// TwinCAT 3 PLC project FMFiles
// Title: FM Files
// Company: FrameworkMonorepo
// ProjectVersion: 0.0.1
// ProgramVersion: 3.1.4024.0
// libraries:
//   FM Common Interfaces, * (FrameworkMonorepo)
//   FM Events, * (FrameworkMonorepo)
//   FM Strings, * (FrameworkMonorepo)
//   Tc2_Standard, * (Beckhoff Automation GmbH)
//   Tc2_System, * (Beckhoff Automation GmbH)
//   Tc2_Utilities, * (Beckhoff Automation GmbH)
// project tree:
//   File/ Directory.TcPOU, File.TcPOU, FileRemover.TcPOU
//   Version/ Global_Version.TcGVL
// (motion and I/O tree: see PLC project fmtypes)
// real-time tasks:
//   TASK BindingTestTask: cycle T#1ms, priority 20, ADS port 350
//   TASK PlcTask: cycle T#1ms, priority 21, ADS port 351
//   TASK PlcTask1: cycle T#1ms, priority 22, ADS port 352
//   TASK PlcTask2: cycle T#1ms, priority 23, ADS port 353
//   TASK MathTestTask: cycle T#1ms, priority 24, ADS port 354
//   TASK TimesTestsTask: cycle T#1ms, priority 25, ADS port 355

// ---- Version/Global_Version.TcGVL
{attribute 'TcGenerated'}
{attribute 'no-analysis'}
{attribute 'linkalways'}
// This function has been automatically generated from the project information.
VAR_GLOBAL CONSTANT
	{attribute 'const_non_replaced'}
	stLibVersion_FM_Files : ST_LibVersion := (iMajor := 0, iMinor := 0, iBuild := 1, iRevision := 0, nFlags := 0, sVersion := '0.0.1');
END_VAR

// ---- File/Directory.TcPOU
FUNCTION_BLOCK Directory
VAR
	creator : FB_CreateDir; // can only create on level of folder
	remover : FB_RemoveDir; // can only remove topmost folder. Not folder with folders.

	listDir : FB_EnumFindFileList;	
	listing : BOOL;
	_ListDone : BOOL;
	checkingFolder : BOOL;
	checkingFileExistence : BOOL;

	page : ARRAY[0..50 - 1] OF ST_FindFileEntry;
	_FileNameList : ARRAY[0..50 - 1] OF T_MaxString;
	_FileExists : BOOL;
	
	filenameForAlarm : T_MaxString;
	createDirectoryErrorTrig : R_TRIG;
	removeDirectoryErrorTrig : R_TRIG;
	listingDirectoryErrorTrig : R_TRIG;
	createDirectoryError : MessageEventLogger(TC_EVENTS.DirectoryEventClass.CreateDirectoryError);
	removeDirectoryError : MessageEventLogger(TC_EVENTS.DirectoryEventClass.RemoveDirectoryError);
	listingDirectoryError : MessageEventLogger(TC_EVENTS.DirectoryEventClass.ListDirectoryError);
END_VAR
VAR CONSTANT
	EntriesPerPage : INT := 50;
END_VAR

METHOD PRIVATE Abort
VAR_INPUT
END_VAR
listDir(
	bExecute := TRUE,
	eCmd := E_EnumCmdType.eEnumCmd_Abort
);
listDir(bExecute := FALSE);
END_METHOD

{attribute 'TcRpcEnable':='1'}
METHOD Create
VAR_INPUT
	path : T_MaxString;
END_VAR
creator(
	sPathName := path,
	bExecute := TRUE,
);
END_METHOD

METHOD Cyclic
VAR
	i : INT;
END_VAR
creator(bExecute := FALSE);
remover(bExecute := FALSE);

listDir(
	pFindList := ADR(page),
	cbFindList := SIZEOF(page)
);

IF (NOT listDir.bBusy AND listing AND NOT _ListDone AND listDir.eCmd <> E_EnumCmdType.eEnumCmd_Abort) THEN

	listDir(bExecute := FALSE);
	listing := FALSE;
	_ListDone := TRUE;
	
	FOR i := 0 TO EntriesPerPage - 1 DO
		_FileNameList[i] := page[i].sFileName;
		
		IF (checkingFileExistence) THEN
			IF (page[i].fileAttributes.bDirectory = checkingFolder
				AND page[i].sFileName <> '') THEN
				_FileExists := TRUE;
			END_IF
		END_IF
	END_FOR
	
	IF (NOT listDir.bEOE) THEN
		Abort();
	END_IF
END_IF

createDirectoryErrorTrig(CLK := creator.bError);
removeDirectoryErrorTrig(CLK := remover.bError);
listingDirectoryErrorTrig(CLK := listDir.bError);

IF (createDirectoryErrorTrig.Q) THEN
	filenameForAlarm := creator.sPathName;
	IF (EventParameters.EscapeBackslash) THEN
		filenameForAlarm := ReplaceAll(filenameForAlarm, '\', '\\'); // Escape backslash to use with web-based HMIs
	END_IF
	createDirectoryError.Arguments.Clear().AddStringByValue(filenameForAlarm);
	createDirectoryError.Send();
END_IF
IF (removeDirectoryErrorTrig.Q) THEN
	filenameForAlarm := remover.sPathName;
	IF (EventParameters.EscapeBackslash) THEN
		filenameForAlarm := ReplaceAll(filenameForAlarm, '\', '\\'); // Escape backslash to use with web-based HMIs
	END_IF
	removeDirectoryError.Arguments.Clear().AddStringByValue(filenameForAlarm);
	removeDirectoryError.Send();
END_IF
IF (listingDirectoryErrorTrig.Q) THEN
	filenameForAlarm := listDir.sPathName;
	IF (EventParameters.EscapeBackslash) THEN
		filenameForAlarm := ReplaceAll(filenameForAlarm, '\', '\\'); // Escape backslash to use with web-based HMIs
	END_IF
	listingDirectoryError.Arguments.Clear().AddStringByValue(filenameForAlarm);
	listingDirectoryError.Send();
END_IF
END_METHOD

{attribute 'monitoring' := 'call'}
PROPERTY FileExists : BOOL
GET
FileExists := _FileExists;
END_GET
END_PROPERTY

{attribute 'monitoring' := 'call'}
PROPERTY FileNameList : REFERENCE TO ARRAY[0..49] OF T_MaxString
GET
FileNameList REF= _FileNameList;
END_GET
END_PROPERTY

METHOD CheckFileExists
VAR_INPUT
	path : T_MaxString;
	folder : BOOL; // FALSE = File, TRUE = Folder
END_VAR
IF (NOT listDir.bBusy) THEN
	
	List(path);
	
	_FileExists := FALSE;
	checkingFileExistence := TRUE;
	checkingFolder := folder;
END_IF
END_METHOD

 // Usage of * wildcard recommended
 // Add * to the end of path to list all files
METHOD List
VAR_INPUT
	path : T_MaxString;
END_VAR
IF (NOT listDir.bBusy) THEN
	
	checkingFileExistence := FALSE;
	listing := TRUE;
	_ListDone := FALSE;
	
	listDir(bExecute := FALSE);
	listDir(
		sPathName := path,
		eCmd := E_EnumCmdType.eEnumCmd_First,
		bExecute := TRUE
	);
END_IF
END_METHOD

PROPERTY ListDone : BOOL
GET
ListDone := _ListDone;
END_GET
END_PROPERTY

METHOD Remove
VAR_INPUT
	path : T_MaxString;
END_VAR
remover(
	sPathName := path,
	bExecute := TRUE,
);
END_METHOD

END_FUNCTION_BLOCK

// ---- File/File.TcPOU
FUNCTION_BLOCK File IMPLEMENTS Cyclic
VAR
	_Busy : BOOL;
	_Done : BOOL;
	_Error : BOOL;
	
	openRequest : BOOL;
	readRequest : BOOL;
	writeRequest : BOOL;
	appendMode : BOOL;
	filePath : T_MaxString;
	
	buffer : POINTER TO BYTE;
	bufferLength : UDINT;

	handle : UINT;
	opener : FB_FileOpen;
	closer : FB_FileClose;
	reader : FB_FileRead;
	writer : FB_FileWrite;
	
	fileState : (Waiting, OpenMode, Opening, Reading, Writing, Closing);
	
	filenameForAlarm : T_MaxString;
	openErrorTrigger : R_TRIG;
	readErrorTrigger : R_TRIG;
	writeErrorTrigger : R_TRIG;
	closeErrorTrigger : R_TRIG;
	notFoundError : MessageEventLogger(TC_EVENTS.FileEventClass.InvalidPath);
	fileOpenError : MessageEventLogger(TC_EVENTS.FileEventClass.OpenFileError);
	fileReadError : MessageEventLogger(TC_EVENTS.FileEventClass.ReadFileError);
	fileWriteError : MessageEventLogger(TC_EVENTS.FileEventClass.WriteFileError);
	fileCloseError : MessageEventLogger(TC_EVENTS.FileEventClass.CloseFileError);
END_VAR
VAR CONSTANT
	NotFoundErrorNumber : UDINT := 16#70C;
END_VAR

{attribute 'monitoring' := 'call'}
PROPERTY Busy : BOOL
GET
Busy := _Busy;
END_GET
END_PROPERTY

METHOD Cyclic
CASE fileState OF
	
	Waiting:
	
		IF (openRequest) THEN
			openRequest := FALSE;
			_Done := FALSE;
			
			fileState := OpenMode;
		END_IF
	
	OpenMode:
	
		IF (readRequest) THEN
			opener.nMode := FOPEN_MODEREAD;
		ELSIF (writeRequest) THEN
			IF (appendMode) THEN
				opener.nMode := FOPEN_MODEAPPEND;
			ELSE
				opener.nMode := FOPEN_MODEWRITE;
			END_IF
		END_IF
		
		opener.nMode := opener.nMode OR FOPEN_MODETEXT;

		fileState := Opening;
	
	Opening:
	
		opener(
			bExecute := NOT opener.bBusy,
			sPathName := filePath,
			hFile => handle,
		);
		
		IF (NOT opener.bExecute AND NOT opener.bBusy AND handle <> 0) THEN
			opener();
			IF (readRequest) THEN
				fileState := Reading;
			ELSIF (writeRequest) THEN
				fileState := Writing;
			END_IF
		END_IF
	
	Reading:
	
		reader(
			bExecute := NOT reader.bBusy,
			hFile := handle,
			pReadBuff := buffer,
			cbReadLen := bufferLength,
		);
		
		IF (NOT reader.bExecute AND NOT reader.bBusy) THEN
			fileState := Closing;
		END_IF
	
	Writing:
	
		writer(
			bExecute := NOT writer.bBusy,
			hFile := handle,
			pWriteBuff := buffer,
			cbWriteLen := bufferLength,
		);
		
		IF (NOT writer.bExecute AND NOT writer.bBusy) THEN
			fileState := Closing;
		END_IF
	
	Closing:
	
		IF (handle = 0) THEN
			fileState := Waiting;
		ELSE
			closer(
				bExecute := NOT closer.bBusy,
				hFile := handle,
			);
			
			IF (NOT closer.bExecute AND NOT closer.bBusy) THEN
				closer();
				handle := 0;
				_Done := TRUE;
				
				fileState := Waiting;
			END_IF
		END_IF
	
END_CASE

_Busy := fileState <> Waiting;

openErrorTrigger(CLK := opener.bError);
readErrorTrigger(CLK := reader.bError);
writeErrorTrigger(CLK := writer.bError);
closeErrorTrigger(CLK := closer.bError);
_Error := 
	openErrorTrigger.Q
	OR readErrorTrigger.Q
	OR writeErrorTrigger.Q
	OR closeErrorTrigger.Q
	;
IF (_Error) THEN
	openRequest := FALSE;
	readRequest := FALSE;
	writeRequest := FALSE;
	
	filenameForAlarm := opener.sPathName;
	IF (EventParameters.EscapeBackslash) THEN
		filenameForAlarm := ReplaceAll(filenameForAlarm, '\', '\\'); // Escape backslash to use with web-based HMIs
	END_IF
	
	IF (openErrorTrigger.Q AND opener.nErrId = NotFoundErrorNumber) THEN
		notFoundError.Arguments.Clear().AddStringByValue(filenameForAlarm);
		notFoundError.Send();
	ELSIF (openErrorTrigger.Q) THEN
		fileOpenError.Arguments.Clear().AddStringByValue(filenameForAlarm);
		fileOpenError.Send();
	ELSIF (readErrorTrigger.Q) THEN
		fileReadError.Arguments.Clear().AddStringByValue(filenameForAlarm);
		fileReadError.Send();
	ELSIF (openErrorTrigger.Q) THEN
		fileWriteError.Arguments.Clear().AddStringByValue(filenameForAlarm);
		fileWriteError.Send();
	ELSIF (openErrorTrigger.Q) THEN
		fileCloseError.Arguments.Clear().AddStringByValue(filenameForAlarm);
		fileCloseError.Send();
	END_IF
	
	IF (fileState > Waiting AND fileState < Closing) THEN
		fileState := Closing;
	END_IF
END_IF
END_METHOD

{attribute 'monitoring' := 'call'}
PROPERTY Done : BOOL
GET
Done := _Done;
END_GET
END_PROPERTY

{attribute 'monitoring' := 'call'}
PROPERTY Error : BOOL
GET
Error := _Error;
END_GET
END_PROPERTY

METHOD Read
VAR_INPUT
	buffer : POINTER TO BYTE;
	bufferLength : UDINT;
	filePath : T_MaxString;
END_VAR
IF (NOT _Busy) THEN
	THIS^.filePath := filePath;
	THIS^.buffer := buffer;
	THIS^.bufferLength := bufferLength;
	
	openRequest := TRUE;
	readRequest := TRUE;
	writeRequest := FALSE;
END_IF
END_METHOD

METHOD Write
VAR_INPUT
	buffer : POINTER TO BYTE;
	bufferLength : UDINT;
	filePath : T_MaxString;
	append : BOOL;
END_VAR
IF (NOT _Busy) THEN
	THIS^.filePath := filePath;
	THIS^.buffer := buffer;
	THIS^.bufferLength := bufferLength;
	
	openRequest := TRUE;
	writeRequest := TRUE;
	readRequest := FALSE;
	appendMode := append;
END_IF
END_METHOD

END_FUNCTION_BLOCK

// ---- File/FileRemover.TcPOU
FUNCTION_BLOCK FileRemover IMPLEMENTS Cyclic
VAR
	remover : FB_FileDelete;
	
	filenameForAlarm : T_MaxString;
	removeErrorTrigger : R_TRIG;
	notFoundError : MessageEventLogger(TC_EVENTS.FileEventClass.InvalidPath);
	removeError : MessageEventLogger(TC_EVENTS.FileEventClass.RemoveFileError);
	
	removing : BOOL;
	_Done : BOOL;
END_VAR
VAR CONSTANT
	NotFoundErrorNumber : UDINT := 16#70C;
END_VAR

{attribute 'monitoring' := 'call'}
PROPERTY Busy : BOOL
GET
Busy := remover.bBusy;
END_GET
END_PROPERTY

METHOD Cyclic
remover(bExecute := FALSE);

IF (NOT remover.bBusy) THEN
	IF (NOT remover.bError AND removing) THEN
		_Done := TRUE;
	END_IF
	removing := FALSE;
END_IF

removeErrorTrigger(CLK := remover.bError);
IF (removeErrorTrigger.Q) THEN
	
	filenameForAlarm := remover.sPathName;
	IF (EventParameters.EscapeBackslash) THEN
		filenameForAlarm := ReplaceAll(filenameForAlarm, '\', '\\'); // Escape backslash to use with web-based HMIs
	END_IF
	
	IF (remover.nErrId = NotFoundErrorNumber) THEN
		notFoundError.Arguments.Clear().AddStringByValue(filenameForAlarm);
		notFoundError.Send();
	ELSE
		removeError.Arguments.Clear().AddStringByValue(filenameForAlarm);
		removeError.Send();
	END_IF
END_IF
END_METHOD

{attribute 'monitoring' := 'call'}
PROPERTY Done : BOOL
GET
Done := _Done;
END_GET
END_PROPERTY

{attribute 'monitoring' := 'call'}
PROPERTY Error : BOOL
GET
Error := remover.bError;
END_GET
END_PROPERTY

METHOD Remove
VAR_INPUT
	filePath : T_MaxString;
END_VAR
removing := TRUE;
_Done := FALSE;

remover(
	sPathName := filePath,
	bExecute := TRUE
);
END_METHOD

END_FUNCTION_BLOCK
